Staubli VAL3: reset.pgx

public program reset(num x_nConvNum (dimensions=1), num& x_nError[] (dimensions=1))
// Reset the tracking libraries without killing every task(s)
begin
  // This program resets the conveyor library
  //
  // Input Param
  //  x_nConvNum  : Number of the conveyor
  //
  // Output Param
  //  x_nError    : Error code
  //    0    --> No error
  //    3    --> Invalid conveyor number
  //
  //----------------------------------------------------------------
  //
  bReset=true
  x_nError=0
  switch x_nConvNum
    case 0
      call cnv0:reset()
    break
    case 1
      call cnv1:reset()
    break
    default
      x_nError=3
    break
  endSwitch
end
